(* IEC 61131-3 sources: Lasal/CPU_5344_V01/Class/CheckCanState, 1 file *)

(* ---- CheckCanState.st ---- *)
(*!
<Class
	Name               = "CheckCanState"
	Revision           = "0.0"
	RealtimeTask       = "false"
	CyclicTask         = "false"
	BackgroundTask     = "false"
	Sigmatek           = "false"
	OSInterface        = "false"
	HighPriority       = "false"
	Automatic          = "false"
	UpdateMode         = "Prescan"
	SharedCommandTable = "true"
	Objectsize         = "(394,120)">
	<Channels>
		<Server Name="ClassSvr" Visualized="false" Initialize="false" WriteProtected="true" Retentive="false"/>
		<Client Name="CanControl1" Required="false" Internal="false"/>
		<Client Name="CanControl2" Required="false" Internal="false"/>
		<Client Name="CanControl3" Required="false" Internal="false"/>
		<Client Name="CanControl4" Required="false" Internal="false"/>
	</Channels>
</Class>
*)
CheckCanState : CLASS
  //Servers:
	ClassSvr 	: SvrChCmd_DINT;
  //Clients:
	CanControl1 	: CltCh_DINT;
	CanControl2 	: CltCh_DINT;
	CanControl3 	: CltCh_DINT;
	CanControl4 	: CltCh_DINT;
  //Variables:
		conCan1 	: DINT;
		conCan2 	: DINT;
		conCan3 	: DINT;
		conCan4 	: DINT;
  //Functions:

	FUNCTION VIRTUAL GLOBAL Init;

	FUNCTION VIRTUAL GLOBAL ClassSvr::Read
		VAR_OUTPUT
			output (EAX) 	: DINT;
		END_VAR;
  //Tables:
	FUNCTION @STD
		VAR_OUTPUT
			ret_code	: CONFSTATES;
		END_VAR;
	FUNCTION GLOBAL TAB @CT_;
END_CLASS;

FUNCTION VIRTUAL GLOBAL CheckCanState::Init

conCan1 := IsClientConnected(input:=#CanControl1);
conCan2 := IsClientConnected(input:=#CanControl2);
conCan3 := IsClientConnected(input:=#CanControl3);
conCan4 := IsClientConnected(input:=#CanControl4);

END_FUNCTION

FUNCTION VIRTUAL GLOBAL CheckCanState::ClassSvr::Read
	VAR_OUTPUT
		output (EAX) 	: DINT;
	END_VAR

  CanControl1 := CanControl1.Read();
  CanControl2 := CanControl2.Read();
  CanControl3 := CanControl3.Read();
  CanControl4 := CanControl4.Read();

  ClassSvr := TRUE;

  if conCan1 = TRUE & CanControl1 <> 1 then
    ClassSvr := FALSE;
  end_if;

  if conCan2 = TRUE & CanControl2 <> 1 then
    ClassSvr := FALSE;
  end_if;

  if conCan3 = TRUE & CanControl3 <> 1 then
    ClassSvr := FALSE;
  end_if;

  if conCan4 = TRUE & CanControl4 <> 1 then
    ClassSvr := FALSE;
  end_if;

	output := ClassSvr;

END_FUNCTION
